TYPE ST_MGMT_ThNTZ_Aktor_Zustand :
STRUCT
	EIN_Anford			: BOOL;
	EIN_Prioritaet			: SINT;
	AUS_Anford			: BOOL;
	AUS_Prioritaet		: SINT;
END_STRUCT
END_TYPE

(* stored: Version 1.1.0.1, ProductVersion 3.1.4024.9
   DUT ST_MGMT_ThNTZ_Aktor_Zustand: Id {3975808b-71a9-4b6a-89b8-68bfbdad8a36} *)
